FUNCTION_BLOCK FB_ControlBox
VAR_INPUT
	bRealControlBox : BOOL;
	eStatus : E_Status;
END_VAR
VAR_OUTPUT
	eMode : E_Mode;
END_VAR
VAR
	fbVirtualControlBox : FB_VirtualControlBox;
	fbRealControlBox : FB_RealControlBox;
	fbSelectedControlBox : I_ControlBox := fbVirtualControlBox;
END_VAR

IF bRealControlBox THEN
	fbSelectedControlBox := fbRealControlBox;
ELSE
	fbSelectedControlBox := fbVirtualControlBox;
END_IF	
	
fbSelectedControlBox.ModeSelector(
	eMode => eMode
);

IF G_Work.eStatus = E_Status.Running THEN
	G_VirtualControlBox.bGreenLight :=  TRUE;
ELSE
	G_VirtualControlBox.bGreenLight :=  FALSE;
END_IF

IF G_Work.eStatus = E_Status.Fault THEN
	G_VirtualControlBox.bRedLight :=  TRUE;
ELSE
	G_VirtualControlBox.bRedLight :=  FALSE;
END_IF

G_Work.fJoystickY := G_VirtualControlBox.fJoystickY;

END_FUNCTION_BLOCK

(* stored: Version 1.1.0.1, ProductVersion 3.1.4024.10
   POU FB_ControlBox: Id {23a5fbb3-746f-49da-9ce4-8057d9ad01ee}, SpecialFunc None *)
